FUNCTION_BLOCK FB_CalcFocalLength2LensSetsMock EXTENDS FB_FalliblePublicMock IMPLEMENTS I_CalcFocalLength2LensSets
VAR
    fbResult : FB_QuantityLREALPublicMock;
END_VAR


METHOD Calculate
VAR_INPUT
    (* Distance from source to downstream lens.*)
    SourceDistance	: I_QuantityLREAL;
    (* Distance between the two lens sets.*)
    DistanceBetween	: I_QuantityLREAL;
    LensSetUpstream	: I_LensSet;
    LensSetDownstream	: I_LensSet;
END_VAR
VAR_IN_OUT
    FocalLength	: FB_QuantityLREALPublic;
END_VAR

FocalLength.Copy(QuantityToCopy := fbResult);
END_METHOD


METHOD SetResult
VAR_INPUT
    Result : FB_QuantityLREALPublicMock;
END_VAR

fbResult := Result;
END_METHOD

END_FUNCTION_BLOCK

(* stored: Version 1.1.0.1
   POU FB_CalcFocalLength2LensSetsMock: Id {50889418-b31a-4aea-939f-345ec0b9796f}, SpecialFunc None
   Method Calculate: Id {f9df9c0c-7e90-45c5-a58c-6f43ae146e2d}
   Method SetResult: Id {200a6f9f-a44c-4baa-a6e4-ab9b2939efbb} *)
